(* IEC 61131-3 sources: VarTools/src/vartools, 3 files *)

(* ---- VarTools.typ ---- *)
(********************************************************************
 * COPYRIGHT --
 ********************************************************************
 * Library: VarInfo
 * File: VarInfo.typ
 * Author: davidblackburn
 * Created: June 02, 2014
 ********************************************************************
 * Data types of library VarInfo
 ********************************************************************)

TYPE
	VAR_ERR_enum :
		(
		VAR_ERR_PV_NOT_FOUND := 14710,
		VAR_ERR_PVITEM_ENUM := 14713,
		VAR_ERR_INVALIDINPUT := 50000,
		VAR_ERR_INVALIDVALUE,
		VAR_ERR_UNSUPPORTEDTYPE,
		VAR_ERR_INVALIDTYPE,
		VAR_ERR_TOO_MANY_ITEMS,
		VAR_ERR_
		);
	VAR_TYPE_enum :
		(
		VAR_TYPE_STRUCT := 0, (*0*)
		VAR_TYPE_BOOL,
		VAR_TYPE_SINT,
		VAR_TYPE_INT,
		VAR_TYPE_DINT,
		VAR_TYPE_USINT, (*5*)
		VAR_TYPE_UINT,
		VAR_TYPE_UDINT,
		VAR_TYPE_REAL,
		VAR_TYPE_STRING,
		VAR_TYPE_ULINT, (*10*)
		VAR_TYPE_DATE_AND_TIME,
		VAR_TYPE_TIME,
		VAR_TYPE_DATE,
		VAR_TYPE_LREAL,
		VAR_TYPE_ARRAY_OF_STRUCT, (*15*)
		VAR_TYPE_TIME_OF_DAY,
		VAR_TYPE_BYTE,
		VAR_TYPE_WORD,
		VAR_TYPE_DWORD,
		VAR_TYPE_LWORD, (*20*)
		VAR_TYPE_WSTRING, (*21*)
		VAR_TYPE_LINT := 23, (*23*)
		VAR_TYPE_UNDEFINED := 999
		);
	varVariable_typ : 	STRUCT
		name : STRING[VAR_STRLEN_NAME];
		value : STRING[VAR_STRLEN_VALUE];
		address : UDINT;
		dataType : UDINT;
		length : UDINT;
		dimension : UINT;
	END_STRUCT;
END_TYPE

(* ---- VarTools.fun ---- *)
(********************************************************************
 * COPYRIGHT --
 ********************************************************************
 * Library: VarInfo
 * File: VarInfo.fun
 * Author: davidblackburn
 * Created: June 02, 2014
 ********************************************************************
 * Functions and function blocks of library VarInfo
 ********************************************************************)

FUNCTION varGetInfo : UINT (*Get variable information*) (*$GROUP=User*)
	VAR_INPUT
		pVariable : UDINT;
	END_VAR
END_FUNCTION

FUNCTION varGetValue : UINT (*Get the value of a variable as a string*) (*$GROUP=User*)
	VAR_INPUT
		pVariable : UDINT;
	END_VAR
END_FUNCTION

FUNCTION varGetLrealValue : UINT (*Get the value of a variable as an lreal*)
	VAR_INPUT
		pVariable : UDINT;
		pValue : UDINT;
	END_VAR
END_FUNCTION

FUNCTION varGetRealValue : UINT (*Get the value of a variable as a real*) (*$GROUP=User*)
	VAR_INPUT
		pVariable : UDINT;
		pValue : UDINT;
	END_VAR
END_FUNCTION

FUNCTION varRefresh : UINT (*Force refresh of variable information in next getValue call*)
	VAR_INPUT
		pVariable : UDINT;
	END_VAR
END_FUNCTION

FUNCTION varSetValue : UINT (*Set the value of a variable from a string*) (*$GROUP=User*)
	VAR_INPUT
		pVariable : UDINT;
	END_VAR
END_FUNCTION

FUNCTION varGetVariableList : UINT (*Get a list of all local and global variables with a given name*) (*$GROUP=User*)
	VAR_INPUT
		pVariableName : UDINT;
		List : UDINT;
	END_VAR
END_FUNCTION

FUNCTION varGetTaskList : UINT (*Get a list of all tasks running on the system*) (*$GROUP=User*)
	VAR_INPUT
		List : STRING[80];
		size : UDINT;
	END_VAR
END_FUNCTION

FUNCTION varPopulateMemberNames : BOOL
	VAR_INPUT
		PVName : STRING[80];
		prefix : USINT;
	END_VAR
END_FUNCTION

FUNCTION_BLOCK varVariableWatch
	VAR_INPUT
		pVariable : {REDUND_UNREPLICABLE} UDINT;
	END_VAR
	VAR_OUTPUT
		Status : UINT;
	END_VAR
	VAR
		iName : STRING[VAR_STRLEN_NAME];
		iValue : STRING[VAR_STRLEN_VALUE];
	END_VAR
END_FUNCTION_BLOCK

FUNCTION_BLOCK variableBrowser (*TODO: Add your comment here*) (*$GROUP=User,$CAT=User,$GROUPICON=User.png,$CATICON=User.png*)
	VAR_INPUT
		VariableName : STRING[VAR_STRLEN_VALUE];
		MemberIndex : INT;
		Back : BOOL;
	END_VAR
	VAR_OUTPUT
		CurrentVariable : STRING[VAR_STRLEN_VALUE];
		MemberName : ARRAY[0..VAR_MAI_MEMBERS] OF STRING[VAR_STRLEN_NAME];
		MemberValue : ARRAY[0..VAR_MAI_MEMBERS] OF STRING[VAR_STRLEN_VALUE];
		MemberInfo : ARRAY[0..VAR_MAI_MEMBERS] OF varVariable_typ;
		NumberMembers : UINT;
		info : varVariable_typ;
	END_VAR
	VAR
		iMemberWatch : ARRAY[0..VAR_MAI_MEMBERS] OF varVariableWatch;
		iCurrentWatch : varVariableWatch;
		iLevel : ARRAY[0..19] OF STRING[32];
		iLevelIndex : USINT;
		iMemberIndex : USINT;
	END_VAR
END_FUNCTION_BLOCK

(* ---- VarTools.var ---- *)
(********************************************************************
 * COPYRIGHT --
 ********************************************************************
 * Library: VarInfo
 * File: VarInfo.var
 * Author: davidblackburn
 * Created: June 02, 2014
 ********************************************************************
 * Constants of library VarInfo
 ********************************************************************)
VAR CONSTANT
	VAR_STRLEN_NAME : USINT := 120;
	VAR_STRLEN_VALUE : USINT := 120;
	VAR_MAI_MEMBERS : UINT := 49;
	VAR_MAI_VARLIST : USINT := 99;
END_VAR
(*Data type limits*)
VAR CONSTANT
	VAR_MIN_SINT : DINT := -128;
	VAR_MAX_SINT : DINT := 127;
	VAR_MIN_INT : DINT := -32768;
	VAR_MAX_INT : DINT := 32767;
	VAR_MIN_DINT : DINT := -2147483647;
	VAR_MAX_DINT : DINT := 2147483647;
	VAR_MIN_USINT : DINT := 0;
	VAR_MAX_USINT : DINT := 255;
	VAR_MIN_UINT : DINT := 0;
	VAR_MAX_UINT : DINT := 65535;
	VAR_MIN_UDINT : UDINT := 0;
	VAR_MAX_UDINT : UDINT := 4294967295;
	VAR_MIN_REAL : REAL := -3.4E038;
	VAR_MAX_REAL : REAL := 3.4E038;
END_VAR
